// TwinCAT 3 PLC project PLC1
// ProgramVersion: 3.1.4024.0
// libraries:
//   Tc2_Standard, * (Beckhoff Automation GmbH)
//   Tc2_System, * (Beckhoff Automation GmbH)
//   Tc2_Utilities, * (Beckhoff Automation GmbH)
//   Tc3_Module, * (Beckhoff Automation GmbH)
// project tree:
//   / PlcTask.TcTTO
//   POUs/ Factorial.TcPOU, MAIN.TcPOU
// real-time tasks:
//   TASK PlcTask: cycle T#10ms, priority 20, ADS port 350

CONFIGURATION PLC1
    RESOURCE PLC ON TwinCAT3
        TASK PlcTask(INTERVAL := T#10ms, PRIORITY := 20);
        PROGRAM MAIN WITH PlcTask : MAIN;
    END_RESOURCE
END_CONFIGURATION

// ---- POUs/MAIN.TcPOU
PROGRAM MAIN
VAR
	Profiler: PROFILER;
	ProfilerResult  : PROFILERSTRUCT;
	nFactorial: ULINT;
END_VAR

Profiler(START:=TRUE,RESET:=TRUE);
Factorial(n:=nFactorial);
Profiler(START:=FALSE);
ProfilerResult:= Profiler.Data;

END_PROGRAM

// ---- POUs/Factorial.TcPOU
FUNCTION Factorial : ULINT
VAR_INPUT
	n: ULINT;
END_VAR
VAR
	nReturnValue: ULINT;
	i: ULINT;
END_VAR

nReturnValue := 1;
FOR i := 1 TO n BY 1 DO
	nReturnValue := nReturnValue * i;
END_FOR
Factorial := nReturnValue;

END_FUNCTION
